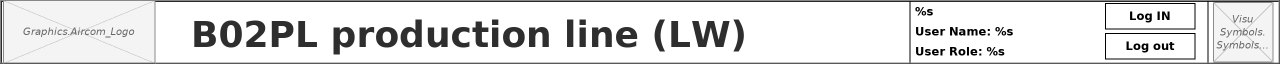
VISUALIZATION TitleBar  // 1280x64
    Rectangle (0,0 1280x64)
    Image (1213,2 60x60), image: VisuSymbols.Symbols.Home
        OnMouseDown: change screen: HomeVisu
        OnMouseDown: FrameSelectionChange Selection=Selection=-1, GlobSel=IndExpr=0, AssignDir=HomeVisu.MainMenu_Frame, AssignType=Directly, SelType=Globally
    Image (3,0 152x63), image: Graphics.Aircom_Logo
    Rectangle (912,2 180x19), "%s", text variable: GVL_Aircom.stAC_DT_Data.sTimeString
    Rectangle (912,22 180x19), "User Name: %s", text variable: GVL.fbUserLogin.sUserName
    Rectangle (912,42 180x19), "User Role: %s", text variable: TO_STRING(GVL.fbUserLogin.nUserRole)
    RoundedRectangle (1105,33 90x26), "Log out", invisible if: NOT GVL.fbUserLogin.bUserLogged
        OnMouseClick: execute { GVL.fbUserLogin.bUserLogged := FALSE; }
        OnMouseClick: FrameSelectionChange Selection=Selection=-1, GlobSel=IndExpr=0, AssignDir=HomeVisu.MainMenu_Frame, AssignType=Directly, SelType=Globally
    Rectangle (1105,3 90x26), "User loged", text variable: GVL.fbUserLogin.sUserName, invisible if: NOT GVL.fbUserLogin.bUserLogged
    Line (910,64) (910,1)
    Line (1208,64) (1208,1)
    RoundedRectangle (1105,3 90x26), "Log IN", invisible if: GVL.fbUserLogin.bUserLogged
        OnMouseClick: write GVL.fbUserLogin.sScanedId via Edit, format %s, password
    Rectangle (188,10 647x49), "B02PL production line (LW)"
END_VISUALIZATION

(* stored: Version 1.1.0.1, ProductVersion 3.1.4024.12
   Visu TitleBar: Id {79f85e50-3093-4006-acf3-c75b6ca88c49} *)
